FUNCTION_BLOCK test
VAR_INPUT
END_VAR
VAR_OUTPUT
END_VAR
VAR
END_VAR

MessageToPublish := 'Kloepfer, Pohle, Wild';
    fbMqttClient.Publish(sTopic:= '$$ names',
		pPayload:= ADR(MessageToPublish),
		nPayloadSize:= LEN(MessageToPublish)+1,
		eQoS:= TcIotMqttQos.AtMostOnceDelivery,
		bRetain:= TRUE,
		bQueue:= FALSE);
			
	MessageToPublish := 'IBK MQTTea Party';
    fbMqttClient.Publish(sTopic:= '$$ groupname',
		pPayload:= ADR(MessageToPublish),
		nPayloadSize:= LEN(MessageToPublish)+1,
		eQoS:= TcIotMqttQos.AtMostOnceDelivery,
		bRetain:= TRUE,
		bQueue:= FALSE);
		
	MessageToPublish := 'meter';
	fbMqttClient.Publish(sTopic:= 'Fuellstand/$$unit',
		pPayload:= ADR(MessageToPublish),
		nPayloadSize:= LEN(MessageToPublish)+1,
		eQoS:= TcIotMqttQos.AtMostOnceDelivery,
		bRetain:= TRUE,
		bQueue:= FALSE);

END_FUNCTION_BLOCK

(* stored: Version 1.1.0.1, ProductVersion 3.1.4024.12
   POU test: Id {c294c721-8aa1-4db4-ad5d-7c9cb24ffc79}, SpecialFunc None *)
